{attribute 'qualified_only'}
{attribute 'strict'}
{attribute 'to_string'}
TYPE PickPlaceSteps :
(
	WaitingForAutomaticStart := 0,
	DriveToHome,
	DriveXYToPick,
	DriveZDown,
	GrabPart,
	DriveZUp
);
END_TYPE

(* stored: Version 1.1.0.1
   DUT PickPlaceSteps: Id {5f2039d2-005d-4c2d-8e20-2159eea26a7f} *)
